// --- N54 D2 Control On add-on logic ---------------------------------------
// "EnableControlOn := BusOk AND NOT ControlOffButtonPressed", then reset by the
// Main/Safety-Valve add-ons on a compressed-air error. Guard doors deliberately
// do NOT gate it: the standard states the add-on still sets EnableControlOn (and
// briefly SwitchControlOn) while doors are open - the relay chain enforces the
// door condition.
EnableControlOn := BusOk AND NOT ControlOffButton AND AirPressureOk;
ControlOffSet   := NOT EnableControlOn;

// SwitchControlOn: exactly two seconds from the button's rising edge, cancelled
// immediately by Control Off (which has priority over Control On).
_onEdge(CLK := ControlOnButton);
IF ControlOffButton OR _switchTimer.Q THEN
    _switchActive := FALSE;
ELSIF _onEdge.Q AND EnableControlOn THEN
    _switchActive := TRUE;
END_IF
_switchTimer(IN := _switchActive, PT := T#2S);
SwitchControlOn := _switchActive;
END_METHOD

END_FUNCTION_BLOCK
